(* Controls all basic machinery in factory *)

PROGRAM Equipment_Controller
  VAR_EXTERNAL
    Safety_OK : BOOL;
    System_Reset : BOOL;
    Conveyor_Start : BOOL;
    Conveyor_Stop : BOOL;
    Ingredient_A_Request : BOOL;
    Ingredient_B_Request : BOOL;
    Discharge_Request : BOOL;
    Packaging_Request : BOOL;
    Mixer_Request : BOOL;
    Conveyor_Fault : BOOL;
    Mixer_Fault : BOOL;
    Packaging_Fault : BOOL;
    Pump_A_Fault : BOOL;
    Pump_B_Fault : BOOL;
    Discharge_Pump_Fault : BOOL;
    Inlet_Valve_Fault : BOOL;
    Ingredient_A_Valve_Fault : BOOL;
    Ingredient_B_Valve_Fault : BOOL;
    Discharge_Valve_Fault : BOOL;
  END_VAR
  VAR
    Conveyor_Motor : FB_Motor;
    Mixer_Motor : FB_Motor;
    Packing_Motor : FB_Motor;
    Pump_A : FB_PUMP;
    Pump_B : FB_PUMP;
    Discharge_Pump : FB_PUMP;
    Inlet_Valve : FB_VALVE;
    Ingredient_A_Valve : FB_VALVE;
    Ingredient_B_Valve : FB_VALVE;
    Discharge_Valve : FB_VALVE;
    Conveyor_Reset : BOOL;
    Conveyor_Fault_In : BOOL;
    Conveyor_Run : BOOL;
    Conveyor_Ready : BOOL;
    Mixer_Start_Cmd : BOOL;
    Mixer_Stop : BOOL;
    Mixer_Reset : BOOL;
    Mixer_Fault_In : BOOL;
    Mixer_Run : BOOL;
    Mixer_Ready : BOOL;
    Packaging_Start : BOOL;
    Packaging_Stop : BOOL;
    Packaging_Reset : BOOL;
    Packaging_Fault_In : BOOL;
    Packaging_Run : BOOL;
    Packaging_Ready : BOOL;
    Pump_A_Start : BOOL;
    Pump_A_Stop : BOOL;
    Pump_A_Reset : BOOL;
    Pump_A_Fault_In : BOOL;
    Pump_A_Run : BOOL;
    Pump_A_Ready : BOOL;
    Pump_B_Start : BOOL;
    Pump_B_Stop : BOOL;
    Pump_B_Reset : BOOL;
    Pump_B_Fault_In : BOOL;
    Pump_B_Run : BOOL;
    Pump_B_Ready : BOOL;
    Discharge_Pump_Start : BOOL;
    Discharge_Pump_Stop : BOOL;
    Discharge_Pump_Reset : BOOL;
    Discharge_Pump_Fault_In : BOOL;
    Discharge_Pump_Run : BOOL;
    Discharge_Pump_Ready : BOOL;
    Inlet_Valve_Open_Cmd : BOOL;
    Inlet_Valve_Close_Cmd : BOOL;
    Inlet_Valve_Fault_In : BOOL;
    Inlet_Valve_Reset : BOOL;
    Inlet_Valve_Open : BOOL;
    Inlet_Valve_Closed : BOOL;
    Ingredient_A_Valve_Open_Cmd : BOOL;
    Ingredient_A_Valve_Close_Cmd : BOOL;
    Ingredient_A_Valve_Fault_In : BOOL;
    Ingredient_A_Valve_Reset : BOOL;
    Ingredient_A_Valve_Open : BOOL;
    Ingredient_A_Valve_Closed : BOOL;
    Ingredient_B_Valve_Open_Cmd : BOOL;
    Ingredient_B_Valve_Close_Cmd : BOOL;
    Ingredient_B_Valve_Fault_In : BOOL;
    Ingredient_B_Valve_Reset : BOOL;
    Ingredient_B_Valve_Open : BOOL;
    Ingredient_B_Valve_Closed : BOOL;
    Discharge_Valve_Open_Cmd : BOOL;
    Discharge_Valve_Close_Cmd : BOOL;
    Discharge_Valve_Fault_In : BOOL;
    Discharge_Valve_Reset : BOOL;
    Discharge_Valve_Open : BOOL;
    Discharge_Valve_Closed : BOOL;
  END_VAR

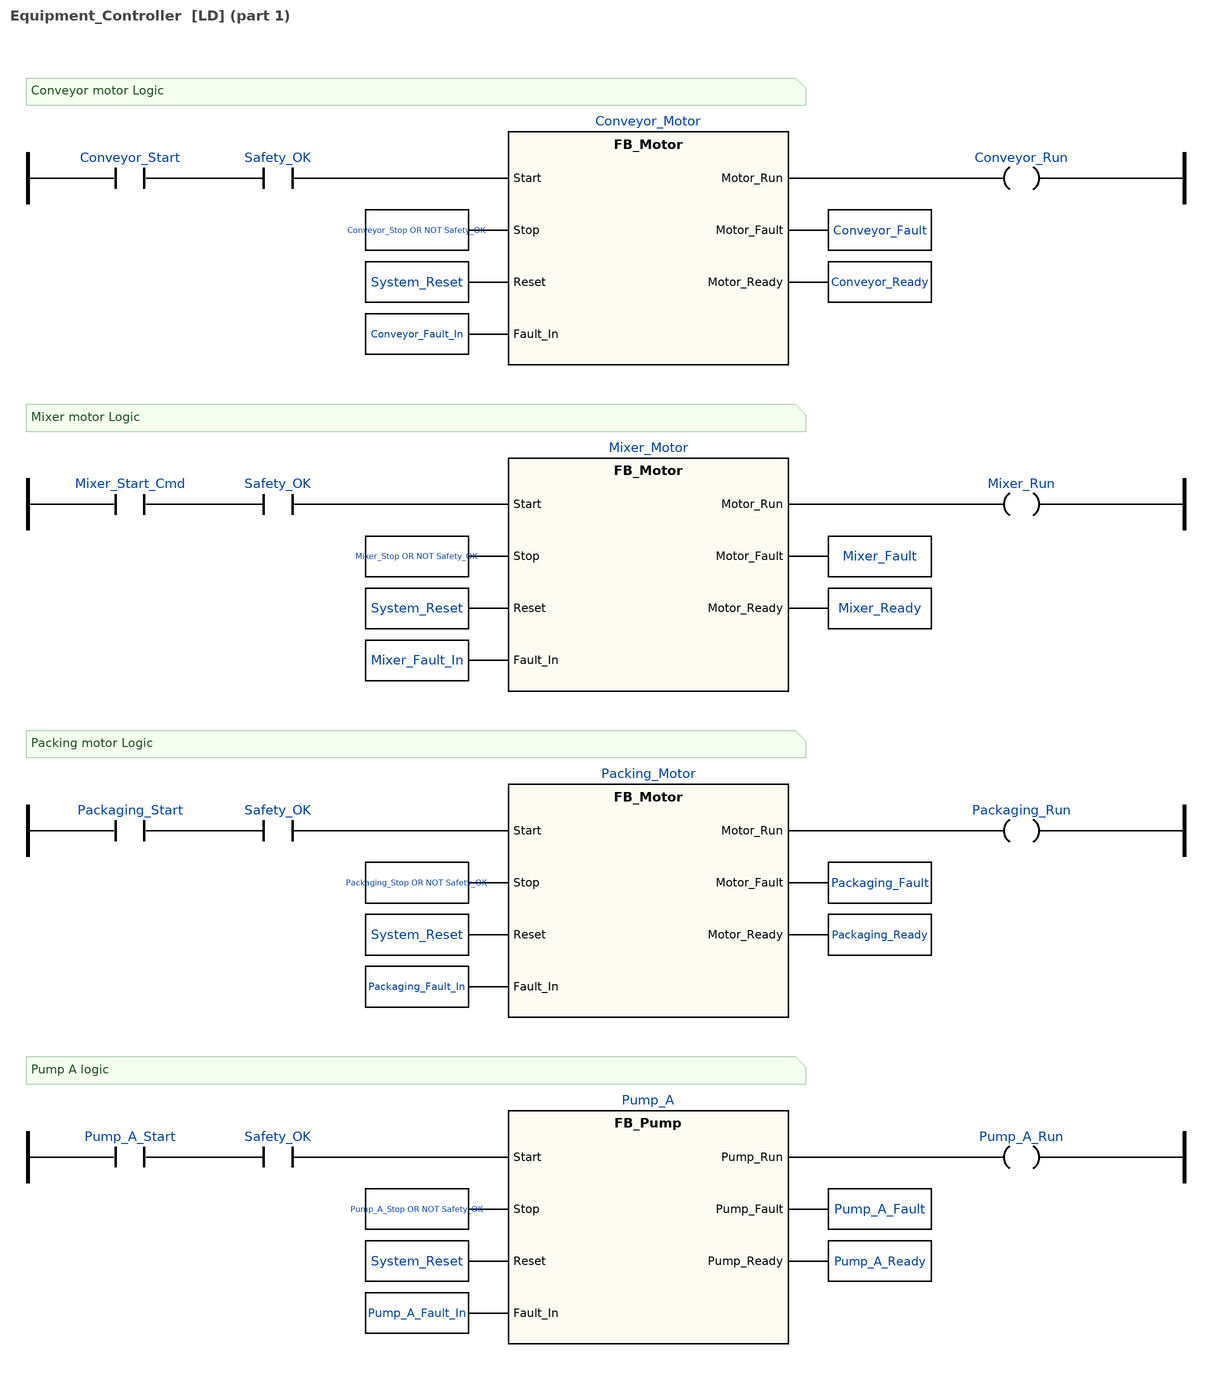
(* LD diagram, written out as Structured Text *)
(* Conveyor motor Logic *)
Conveyor_Motor(Start := Conveyor_Start AND Safety_OK, Stop := Conveyor_Stop OR NOT Safety_OK, Reset := System_Reset, Fault_In := Conveyor_Fault_In);
Conveyor_Run := Conveyor_Motor.Motor_Run;
Conveyor_Fault := Conveyor_Motor.Motor_Fault;
Conveyor_Ready := Conveyor_Motor.Motor_Ready;
(* Mixer motor Logic *)
Mixer_Motor(Start := Mixer_Start_Cmd AND Safety_OK, Stop := Mixer_Stop OR NOT Safety_OK, Reset := System_Reset, Fault_In := Mixer_Fault_In);
Mixer_Run := Mixer_Motor.Motor_Run;
Mixer_Fault := Mixer_Motor.Motor_Fault;
Mixer_Ready := Mixer_Motor.Motor_Ready;
(* Packing motor Logic *)
Packing_Motor(Start := Packaging_Start AND Safety_OK, Stop := Packaging_Stop OR NOT Safety_OK, Reset := System_Reset, Fault_In := Packaging_Fault_In);
Packaging_Run := Packing_Motor.Motor_Run;
Packaging_Fault := Packing_Motor.Motor_Fault;
Packaging_Ready := Packing_Motor.Motor_Ready;
(* Pump A logic *)
Pump_A(Start := Pump_A_Start AND Safety_OK, Stop := Pump_A_Stop OR NOT Safety_OK, Reset := System_Reset, Fault_In := Pump_A_Fault_In);
Pump_A_Run := Pump_A.Pump_Run;
Pump_A_Fault := Pump_A.Pump_Fault;
Pump_A_Ready := Pump_A.Pump_Ready;
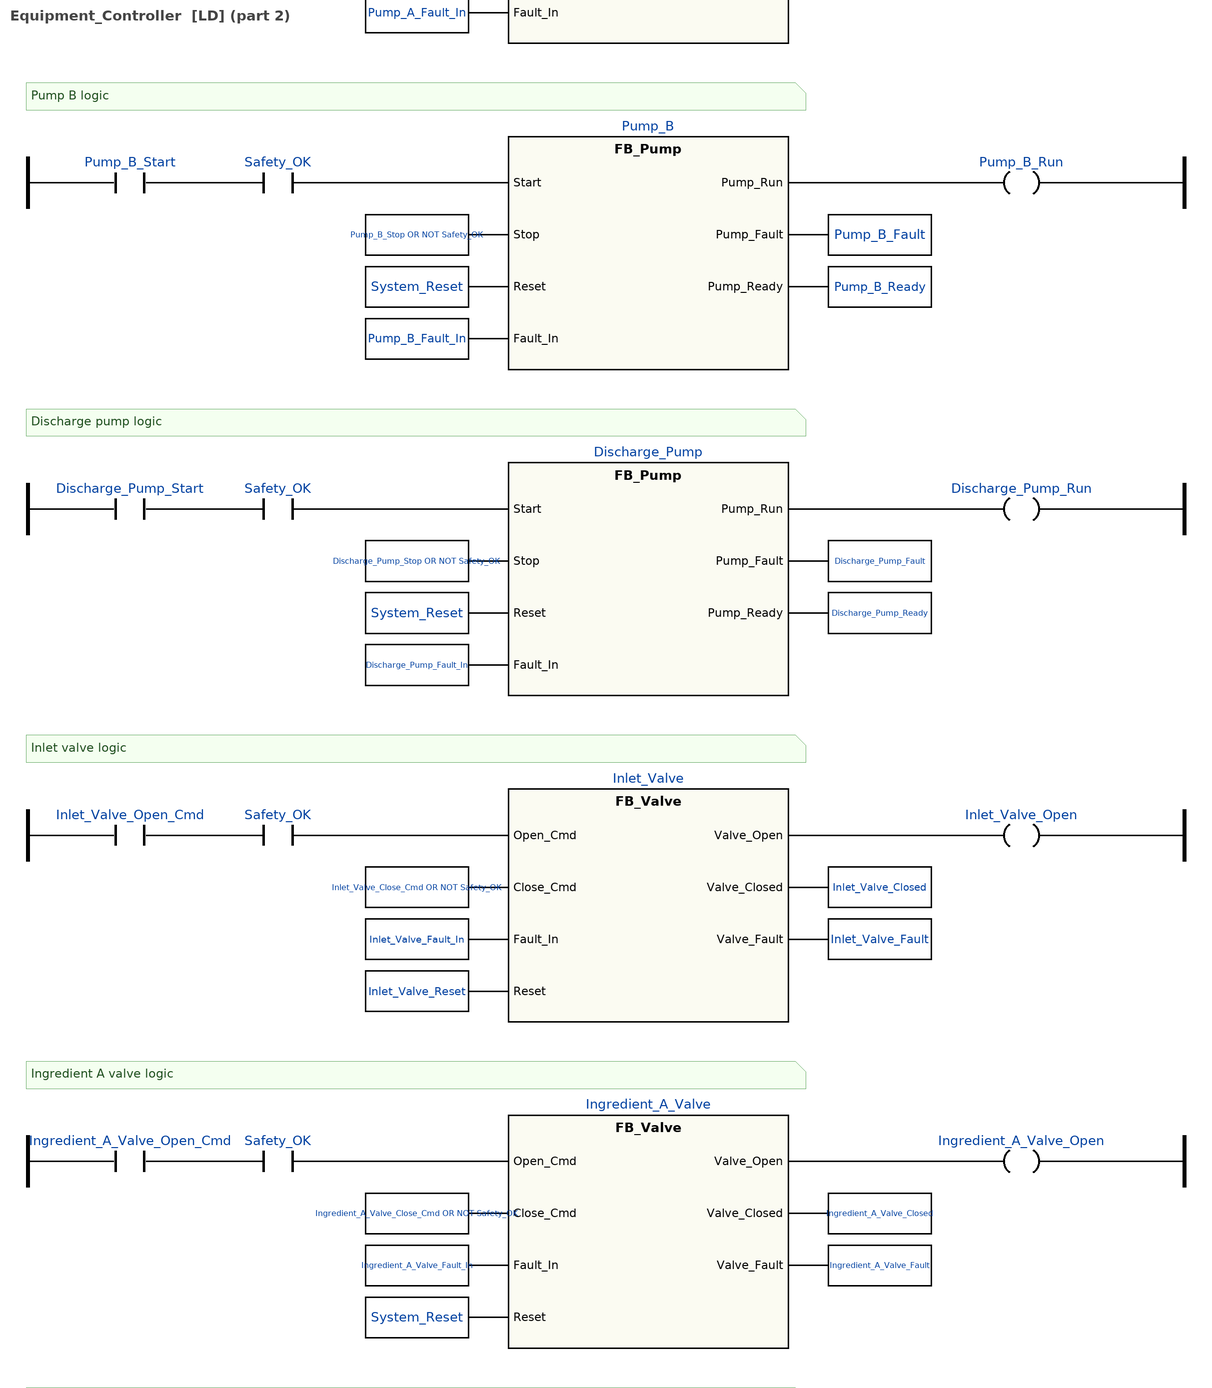
(* Pump B logic *)
Pump_B(Start := Pump_B_Start AND Safety_OK, Stop := Pump_B_Stop OR NOT Safety_OK, Reset := System_Reset, Fault_In := Pump_B_Fault_In);
Pump_B_Run := Pump_B.Pump_Run;
Pump_B_Fault := Pump_B.Pump_Fault;
Pump_B_Ready := Pump_B.Pump_Ready;
(* Discharge pump logic *)
Discharge_Pump(Start := Discharge_Pump_Start AND Safety_OK, Stop := Discharge_Pump_Stop OR NOT Safety_OK, Reset := System_Reset, Fault_In := Discharge_Pump_Fault_In);
Discharge_Pump_Run := Discharge_Pump.Pump_Run;
Discharge_Pump_Fault := Discharge_Pump.Pump_Fault;
Discharge_Pump_Ready := Discharge_Pump.Pump_Ready;
(* Inlet valve logic *)
Inlet_Valve(Open_Cmd := Inlet_Valve_Open_Cmd AND Safety_OK, Close_Cmd := Inlet_Valve_Close_Cmd OR NOT Safety_OK, Fault_In := Inlet_Valve_Fault_In, Reset := Inlet_Valve_Reset);
Inlet_Valve_Open := Inlet_Valve.Valve_Open;
Inlet_Valve_Closed := Inlet_Valve.Valve_Closed;
Inlet_Valve_Fault := Inlet_Valve.Valve_Fault;
(* Ingredient A valve logic *)
Ingredient_A_Valve(Open_Cmd := Ingredient_A_Valve_Open_Cmd AND Safety_OK, Close_Cmd := Ingredient_A_Valve_Close_Cmd OR NOT Safety_OK, Fault_In := Ingredient_A_Valve_Fault_In, Reset := System_Reset);
Ingredient_A_Valve_Open := Ingredient_A_Valve.Valve_Open;
Ingredient_A_Valve_Closed := Ingredient_A_Valve.Valve_Closed;
Ingredient_A_Valve_Fault := Ingredient_A_Valve.Valve_Fault;
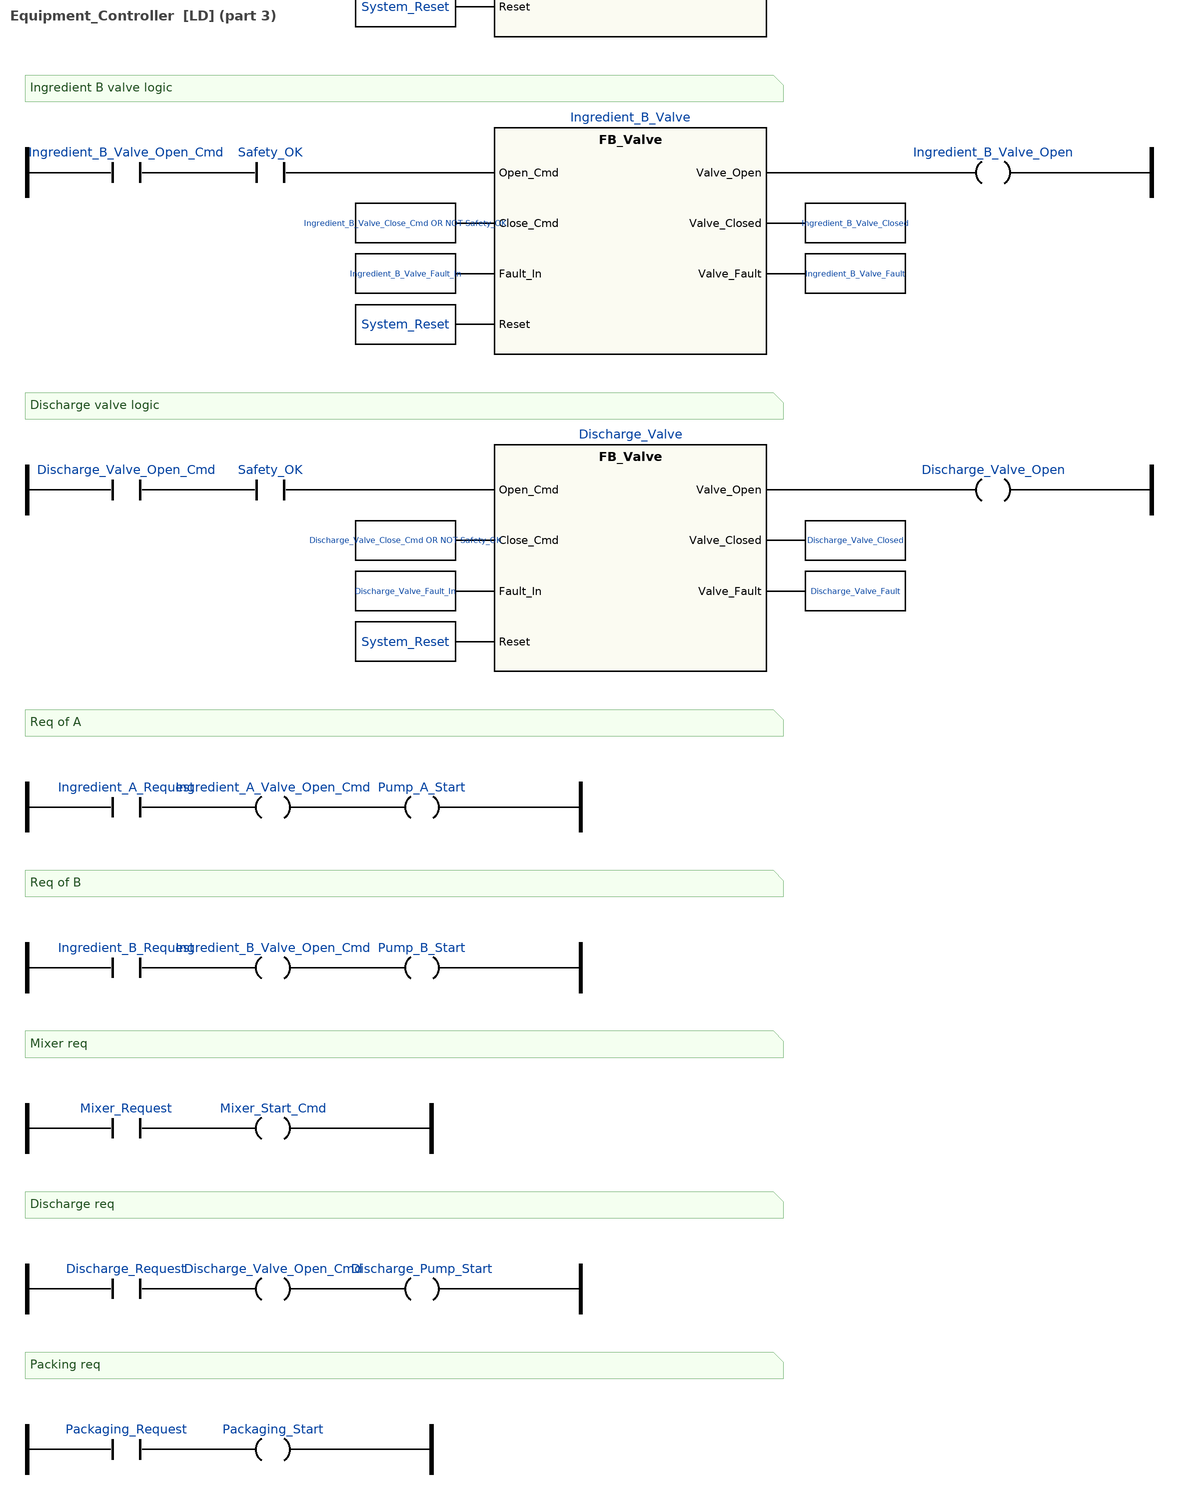
(* Ingredient B valve logic *)
Ingredient_B_Valve(Open_Cmd := Ingredient_B_Valve_Open_Cmd AND Safety_OK, Close_Cmd := Ingredient_B_Valve_Close_Cmd OR NOT Safety_OK, Fault_In := Ingredient_B_Valve_Fault_In, Reset := System_Reset);
Ingredient_B_Valve_Open := Ingredient_B_Valve.Valve_Open;
Ingredient_B_Valve_Closed := Ingredient_B_Valve.Valve_Closed;
Ingredient_B_Valve_Fault := Ingredient_B_Valve.Valve_Fault;
(* Discharge valve logic *)
Discharge_Valve(Open_Cmd := Discharge_Valve_Open_Cmd AND Safety_OK, Close_Cmd := Discharge_Valve_Close_Cmd OR NOT Safety_OK, Fault_In := Discharge_Valve_Fault_In, Reset := System_Reset);
Discharge_Valve_Open := Discharge_Valve.Valve_Open;
Discharge_Valve_Closed := Discharge_Valve.Valve_Closed;
Discharge_Valve_Fault := Discharge_Valve.Valve_Fault;
(* Req of A *)
Ingredient_A_Valve_Open_Cmd := Ingredient_A_Request;
Pump_A_Start := Ingredient_A_Request;
(* Req of B *)
Ingredient_B_Valve_Open_Cmd := Ingredient_B_Request;
Pump_B_Start := Ingredient_B_Request;
(* Mixer req *)
Mixer_Start_Cmd := Mixer_Request;
(* Discharge req *)
Discharge_Valve_Open_Cmd := Discharge_Request;
Discharge_Pump_Start := Discharge_Request;
(* Packing req *)
Packaging_Start := Packaging_Request;
END_PROGRAM
